Staubli VAL3: OnF1.pgx

program OnF1()
  local bool l_bRes
begin

  switch nPage
    case 0
      //编辑路径
      call EditMain(sItem)
    break
    case 1
      //
      tTool.trsf=Tool:tTool[prd:sToolName].trsf
      fFrame.trsf=Frame:fFrame[prd:sFrameName].trsf
      pTemp=here(tTool,fFrame)
      prd:pDemo[nSelected].trsf=pTemp.trsf
    break
    case 2
      //开始


    break
    case 3
    break
    case 4
    break

  endSwitch
end
